(* CoDeSys 2.3 export: PRZEDPOKOJ_PIETRO.EXP *)

(* POU Rooms/Przedpokoj_pietro, ST *)
FUNCTION_BLOCK Przedpokoj_pietro
VAR
	mainLamp:OnOff;
	tmp: BOOL;
END_VAR
mainLamp(input:=H11_1a OR P7_1a OR P8_1a);
P1_1:= mainLamp.state;
P3_1:=mainLamp.state;
END_FUNCTION_BLOCK
